FUNCTION_BLOCK FB_PWM
VAR_INPUT
	tHightime	: TIME;
	tLowtime	: TIME;

END_VAR
VAR_OUTPUT
	output		: BOOL;
END_VAR
VAR
 	timer 		: Tc2_Standard.TON;
	step		: INT;
END_VAR


CASE step OF
	0:	//low
		output:=FALSE;
		timer(IN:=TRUE , PT:=tLowtime , Q=> , ET=> );
		IF timer.Q THEN
			timer(IN:=FALSE);
			step:=1;
		END_IF
		
	1: 	//high
		output:=True;
		timer(IN:=TRUE , PT:=tHightime , Q=> , ET=> );
		IF timer.Q THEN
			timer(IN:=FALSE);
			step:=0;
		END_IF
END_CASE

END_FUNCTION_BLOCK

(* stored: Version 1.1.0.1, ProductVersion 3.1.4020.12
   POU FB_PWM: Id {77f8bac4-ab23-454d-9283-cd639a623d42}, SpecialFunc None *)
